// TIA Portal V17 export
// export: Created 2025-03-05T07:59:01.1711163Z, ExportSetting WithDefaults, DisplayName Totally Integrated Automation Portal, DisplayVersion V17 Update 8, DisplayName TIA Portal Openness, DisplayVersion V17 Update 8, DisplayName TIA Portal Version Control Interface, DisplayVersion V17, DisplayName SINAMICS Startdrive Advanced, DisplayVersion V17 SP2, DisplayName SINAMICS Startdrive G110M, G120, G120C, G120D, G120P, G115D, DisplayVersion V17 SP2, DisplayName SINAMICS Startdrive G130, G150, S120, S150, SINAMICS MV, S210, DisplayVersion V17 SP2, DisplayName STEP 7 Professional, DisplayVersion V17 Update 8, DisplayName SINUMERIK ONE STEP 7 Toolbox, DisplayVersion V17 Update 12, DisplayName SINUMERIK 840D sl STEP 7 Toolbox, DisplayVersion V17 Update 12, DisplayName STEP 7 Safety, DisplayVersion V17 Update 6, DisplayName WinCC Advanced, DisplayVersion V17 Update 8
FUNCTION "FC2432_FULL_DEPTHS_UNIT_03" : Void   // FC2432, LAD
{ S7_Optimized_Access := 'FALSE' }
AUTHOR : ETXETAR
VERSION : 1.0
// Fixture 1 and Fixture 3 will do Face A
// Fixture 2 and Fixture 4 will do Face B
// stored: AutoNumber false, IsIECCheckEnabled false, SetENOAutomatically false, UDAEnableTagReadback false
   VAR_TEMP   // added for the SCL form of the ladder/FBD networks
      _w1 : Bool;
   END_VAR
BEGIN

REGION Network 1: <<<<<<<<<<<<<<<<<<<<< UNIT 03>>>>>>>>>>>>>>>>>>>>>
END_REGION

REGION Network 2: <<<<<<<<<<<<<<<<<<<< FIXTURE 1 >>>>>>>>>>>>>>>>>>>>
END_REGION

REGION Network 3: UNIT 03 FIXTURE 1 STATION 1 FULL DEPTH / FULL DEPTH 1 PULSE
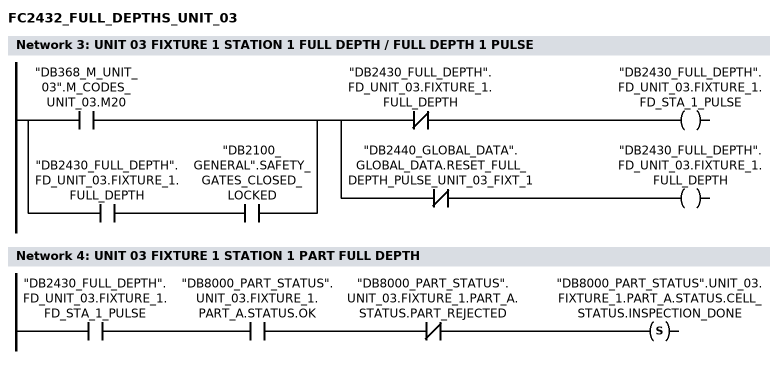
   RUNG wire#powerrail
      Contact( "DB368_M_UNIT_03".M_CODES_UNIT_03.M20 )
      wire#w1
      I_Contact( "DB2430_FULL_DEPTH".FD_UNIT_03.FIXTURE_1.FULL_DEPTH )
      Coil( "DB2430_FULL_DEPTH".FD_UNIT_03.FIXTURE_1.FD_STA_1_PULSE )
   END_RUNG
   RUNG wire#powerrail
      Contact( "DB2430_FULL_DEPTH".FD_UNIT_03.FIXTURE_1.FULL_DEPTH )
      Contact( "DB2100_GENERAL".SAFETY_GATES_CLOSED_LOCKED )
   END_RUNG wire#w1
   RUNG wire#w1
      I_Contact( "DB2440_GLOBAL_DATA".GLOBAL_DATA.RESET_FULL_DEPTH_PULSE_UNIT_03_FIXT_1 )
      Coil( "DB2430_FULL_DEPTH".FD_UNIT_03.FIXTURE_1.FULL_DEPTH )
   END_RUNG
   // the same network as SCL:
   #_w1 := "DB368_M_UNIT_03".M_CODES_UNIT_03.M20 OR ("DB2430_FULL_DEPTH".FD_UNIT_03.FIXTURE_1.FULL_DEPTH AND "DB2100_GENERAL".SAFETY_GATES_CLOSED_LOCKED);
   "DB2430_FULL_DEPTH".FD_UNIT_03.FIXTURE_1.FD_STA_1_PULSE := #_w1 AND NOT "DB2430_FULL_DEPTH".FD_UNIT_03.FIXTURE_1.FULL_DEPTH;
   "DB2430_FULL_DEPTH".FD_UNIT_03.FIXTURE_1.FULL_DEPTH := #_w1 AND NOT "DB2440_GLOBAL_DATA".GLOBAL_DATA.RESET_FULL_DEPTH_PULSE_UNIT_03_FIXT_1;
END_REGION

REGION Network 4: UNIT 03 FIXTURE 1 STATION 1 PART FULL DEPTH
   RUNG wire#powerrail
      Contact( "DB2430_FULL_DEPTH".FD_UNIT_03.FIXTURE_1.FD_STA_1_PULSE )
      Contact( "DB8000_PART_STATUS".UNIT_03.FIXTURE_1.PART_A.STATUS.OK )
      I_Contact( "DB8000_PART_STATUS".UNIT_03.FIXTURE_1.PART_A.STATUS.PART_REJECTED )
      S_Coil( "DB8000_PART_STATUS".UNIT_03.FIXTURE_1.PART_A.STATUS.CELL_STATUS.INSPECTION_DONE )
   END_RUNG
   // the same network as SCL:
   IF "DB2430_FULL_DEPTH".FD_UNIT_03.FIXTURE_1.FD_STA_1_PULSE AND "DB8000_PART_STATUS".UNIT_03.FIXTURE_1.PART_A.STATUS.OK AND NOT "DB8000_PART_STATUS".UNIT_03.FIXTURE_1.PART_A.STATUS.PART_REJECTED THEN
       "DB8000_PART_STATUS".UNIT_03.FIXTURE_1.PART_A.STATUS.CELL_STATUS.INSPECTION_DONE := TRUE;
   END_IF;
END_REGION
END_FUNCTION
